FUNCTION_BLOCK FB_CompressorSystem EXTENDS FB_SystemContinous
VAR_INPUT
END_VAR
VAR_OUTPUT
END_VAR
VAR
	//default parameters
	localDefaultParameters : ST_CompressorDefaultParameters;	

	//pumps
	stPU251DefaultParameters : ST_PumpGrundfosMagna3DefaultParameters := (bPumpBeforeApplication := FALSE, tTaskCycleTime := GlobalVariables.tTaskCycleTime_MAIN, tCtrlCycleTime := GlobalVariables.tCtrlCycleTime_MAIN);
	PU251 : FB_PumpGrundfosMagna3 := (ST_DefaultParameters := stPU251DefaultParameters);;

	//valves
	stRV251DefaultParameters : ST_MixingValveDefaultParameters := (bFeedbackSignal := TRUE, tTaskCycleTime := GlobalVariables.tTaskCycleTime_MAIN, tCtrlCycleTime := GlobalVariables.tCtrlCycleTime_MAIN);		
	RV251 : FB_MixingValve := (ST_DefaultParameters := stRV251DefaultParameters);
	WMZ251 : FB_MollineC3HeatCounter();
		
	//internal variables
	bSetStatusOn_PU251 : BOOL;
	bSetStatusOn_RV251 : BOOL;
END_VAR

MAIN();

PU251.GetState_Profibus();
PU251(bSetStatusOnAutomatic := bSetStatusOn_PU251,
	bAlgorithmPermission := bAlgorithmPermission,
	fSetPointAutomatic := 100,
	nControlModeAutomatic := 0);
PU251.SetState_Profibus();

RV251.GetState_AI();
RV251(bSetStatusOnAutomatic := bSetStatusOn_RV251,
	fSetPointAutomatic := fSetPoint,
	bAlgorithmPermission := bAlgorithmPermission,
	nControlModeAutomatic := 2,
	fTemperatureExternal := PU251.fTemperatureInternal);
RV251.SetState_AO();

WMZ251(aHeatCounterTelegramm := Telegramm_WZ_Druckluftkompressor);

METHOD PROTECTED  CheckError : BOOL
VAR_INPUT
END_VAR
VAR_OUTPUT
	bError : BOOL;
END_VAR
bError := PU251.bError;
END_METHOD

METHOD PROTECTED  Operational : BOOL
VAR_INPUT
END_VAR
VAR_OUTPUT
	bSwitchToWorking : BOOL := FALSE;
END_VAR
bSetStatusOn_PU251 := TRUE;

IF PU251.bStatusOn THEN
	bSwitchToWorking := TRUE;
END_IF
END_METHOD

METHOD PROTECTED  RampDown : BOOL
VAR_INPUT
END_VAR
VAR_OUTPUT
	bRampDownFinished : BOOL := FALSE;
END_VAR
bSetStatusOn_PU251 := FALSE;

IF NOT PU251.bStatusOn THEN
	bSetStatusOn_RV251 := FALSE;
END_IF
END_METHOD

METHOD PROTECTED  RampUp : BOOL
VAR_INPUT
END_VAR
VAR_OUTPUT
	bRampUpFinished : BOOL := FALSE;
END_VAR
bSetStatusOn_RV251 := TRUE;
bRampUpFinished := TRUE;
END_METHOD

METHOD PROTECTED   SetSetPointLimits : BOOL
VAR_INPUT
END_VAR
aSetPointLimits[1] := localDefaultParameters.aSetPointLimitsTemperature[1];
aSetPointLimits[2] := localDefaultParameters.aSetPointLimitsTemperature[2];
END_METHOD

METHOD PROTECTED  SetState : BOOL
VAR_INPUT
END_VAR
VAR_OUTPUT
END_VAR
fOperatingPoint := PU251.fTemperatureInternal;

controlState.bStatusOn := bSetStatusOn;
setPointState.aSetPointLimits := aSetPointLimits;
setPointState.fSetPoint := fSetPoint;
setPointState.fOperatingPoint := fOperatingPoint;
setPointState.sSetPointUnit := 'degreeC';
setPointState.sOperatingPointUnit := 'degreeC';
END_METHOD

METHOD PROTECTED  Working : BOOL
VAR_INPUT
END_VAR
VAR_OUTPUT
	bSwitchToOperational : BOOL := FALSE;
END_VAR
//empty method
END_METHOD

END_FUNCTION_BLOCK

(* stored: Version 1.1.0.1, ProductVersion 3.1.4024.10
   POU FB_CompressorSystem: Id {f1ebdf52-4f03-411c-891c-78a828956cdb}, SpecialFunc None
   Method CheckError: Id {a50d96bf-b53c-410c-87ec-21ce553724aa}
   Method Operational: Id {95b8175c-5301-41c1-a171-418f9517d262}
   Method RampDown: Id {1c464285-ee40-45d5-a501-217e65b5dfe4}
   Method RampUp: Id {4fad2cc8-7e83-4f5b-b8ff-1f31a747421b}
   Method SetSetPointLimits: Id {bcfed1d8-5bc9-4091-8c64-01376c2fe2e2}
   Method SetState: Id {d085a239-6d40-43a4-b7c0-974005529a48}
   Method Working: Id {83ed2a3d-e742-4d4a-be9e-367c734d4463} *)
